Staubli VAL3: readMe.pgx

public program readMe()
begin
  //变换矩阵与转角、通用轴之间的转换
  //
  //addon:motion
end
